Universal Robots PolyScope program: KeyenceRobotVisionSample.urp

Program KeyenceRobotVisionSample (createdIn=3.2.20175 lastSavedIn=3.2.20175 directory=/programs/usbdisk/SampleProgram installation=default robotSerialNumber=2016352004)
Calibrated DH parameters: a=[0.000288, -0.062889, -0.379853, -0.000045, 0.000077, 0]; d=[0.089488, 549.480804, -584.850573, 35.480024, 0.094976, 0.082479]; alpha=[1.570477, -0.000766, -0.002798, 1.569864, -1.570548, 0]; deltaTheta=[-0.000085, -1.422422, 1.677262, -0.254837, -6.283201, 0.00005]
BeforeStart
  Script file /programs/usbdisk/SampleProgram/Sample.script
    | #  This program is a sample program for line operation.
    | #  When using it, please verify the actual operation of the robot
    | #  and make the necessary changes first before implementation.
    | 
    | def CUR_SetUpCamera(CAM, IP_Address, Port):
    | # Pass parameters to global variables.
    |   global Camera = CAM
    |   varmsg("Camera", Camera)
    | 
    |   global IP = IP_Address
    |   varmsg("IP", IP)
    | 
    |   global TelPort = Port
    |   varmsg("TelPort", TelPort)
    | 
    | end
    | 
    | 
    | def CUR_InitComm(CAM):
    | # Open the connection.
    |   global connected = False
    |   while (not  connected):
    |     global connected = socket_open(IP, TelPort, Camera)	# Establish connection to camera
    |     varmsg("connected", connected)						# server via Telnet
    |   end
    |   return connected
    | end
    | 
    | def CUR_TriggImage(CAM):
    | # Send a trigger command.
    |   global Camera = CAM
    |   varmsg("Camera", Camera)
    |   socket_send_string("T1", Camera)			# Set Event and Wait; Acquisition Command
    |   socket_send_byte(13, Camera)				# Carriage Return 0Dhex 13dec
    |   socket_send_byte(10, Camera)				# Line Feed 0Ahex 10dec
    |   global React = socket_read_string(Camera)	# Read answer from camera
    |   varmsg("React", React)
    |   sleep(1.0)
    |   global PositionFromCamera = socket_read_ascii_float(8, Camera)
    |   varmsg("PositionFromCamera", PositionFromCamera)
    | # Wait for the reply.
    |   global posX = PositionFromCamera[2] / 1000
    |   global posY = PositionFromCamera[3] / 1000
    |   global posZ = PositionFromCamera[4] / 1000
    |   global angX = d2r(PositionFromCamera[5])
    |   global angY = d2r(PositionFromCamera[6])
    |   global angZ = d2r(PositionFromCamera[7])
    |   global VisionPos = p[posX, posY, posZ, angX, angY, angZ]
    |   if PositionFromCamera[0] != 8:
    |     return 1
    |   elif PositionFromCamera[1] != 0:
    |     return 2
    |   end
    |   return 0
    | end
    | 
    | 
    | def CUR_Move():
    | # Move to the specified position.
    |   varmsg("VisionPos", VisionPos)
    |   local RealAccel = 0.1
    |   local RealSpeed = 0.1
    | 
    |   A = RPY_to_AxisAngle(VisionPos)
    |   movel(A, RealAccel, RealSpeed)
    | end
    | 
    | def RPY_to_AxisAngle(R):
    | # Conversion (RPY to AxisAngle)
    |   Rx = R[3] / 2.0
    |   Ry = R[4] / 2.0
    |   Rz = R[5] / 2.0
    | 
    |   Cx = cos(Rx)
    |   Sx = sin(Rx)
    |   Cy = cos(Ry)
    |   Sy = sin(Ry)
    |   Cz = cos(Rz)
    |   Sz = sin(Rz)
    | 
    |   Angle = 2.0 * acos(Cx*Cy*Cz + Sx*Sy*Sz)
    |   x = Sx*Cy*Cz - Cx*Sy*Sz
    |   y = Cx*Sy*Cz + Sx*Cy*Sz
    |   z = -Sx*Sy*Cz + Cx*Cy*Sz
    |   Norm = sqrt(x*x + y*y + z*z)
    |   Ratio = Angle / Norm
    |   Ax = x * Ratio
    |   Ay = y * Ratio
    |   Az = z * Ratio
    |   Ans = p[R[0], R[1], R[2], Ax, Ay, Az]
    | 
    |   return Ans
    | end
    | 
    | def CUR_CloseComm(CAM):
    | # Close the connection.
    |   global Camera = CAM
    |   varmsg("Camera", Camera)
    |   socket_close(Camera)
    | end
  Script: CUR_SetUpCamera("Cam1", "192.168.0.10", 8500)
  If CUR_InitComm("Cam1")==False
    Popup Error (haltProgram=false message=Communication Lost)
Robot Program (runOnlyOnce=false motionType=MoveJ speed=1.047198 acceleration=1.396263 recalculateMotions=false)
  triggerResult := CUR_TriggImage("Cam1")   [initializeExpression=0]
  If triggerResult==1
    Popup Error (haltProgram=false message=Communication Error)
  If triggerResult==2
    Popup Error (haltProgram=false message=Search Error)
  Script: CUR_Move()
  Script: CUR_CloseComm("Cam1")
  Halt
